// TIA Portal V17 export
// export: Created 2023-12-05T13:40:22.7138877Z, ExportSetting WithDefaults, DisplayName Totally Integrated Automation Portal, DisplayVersion V17, DisplayName TIA Portal Openness, DisplayVersion V17, DisplayName TIA Portal Version Control Interface, DisplayVersion V17, DisplayName SINAMICS Startdrive Advanced, DisplayVersion V17, DisplayName SINAMICS Startdrive G130, G150, S120, S150, SINAMICS MV, S210, DisplayVersion V17, DisplayName SINAMICS Startdrive G110M, G120, G120C, G120D, G120P, G115D, DisplayVersion V17, DisplayName STEP 7 Professional, DisplayVersion V17, DisplayName STEP 7 Safety, DisplayVersion V17, DisplayName WinCC Professional, DisplayVersion V17
FUNCTION "FC531 ACSPN_V5_1_7 Alarms" : Void   // FC531, LAD
{ S7_Optimized_Access := 'TRUE' }
VERSION : 0.1
// LG 16.03.2023 => Changed Slug sensor ON constantly on unit
// LG 30.06.2022 => Changed name of the block (structures are the same like in STD Block V 5_1_6)
// 07.05.2020 => added copying of one alarm from unit IDB (Address DBX74.6) which is new in SB V_5_1_0
// 10.06.2020 => delete 2byte spare (load dbx74.0 to dbx2.0 etc.)
// 08.09.2021 => Changed name of the block (structures are the same like in STD Block V 5_1_0)
// stored: AutoNumber false, IsIECCheckEnabled false, SetENOAutomatically false, UDAEnableTagReadback false
   VAR_INPUT
      "SB DB" : Int;
      "Alarm DB" : Int;
      "Alarm Offset" : Int;
   END_VAR
   VAR_TEMP
      "SB DBW" : Word;
      "AL DBW" : Word;
      "TR DBW" : Word;
   END_VAR
BEGIN

NETWORK
TITLE = Initialization
      L     #"SB DB";
      T     #"SB DBW";
      L     #"Alarm DB";
      T     #"AL DBW";
      L     #"Alarm Offset";
      SLD   3;
      LAR1;

NETWORK
TITLE = Cylinder faults
      CLR;
      OPN   DB [#"SB DBW"];
      L     %DBB70;
      OPN   DB [#"AL DBW"];
      T     DBB [AR1, P#0.0];

NETWORK
TITLE = Cylinder faults
      CLR;
      OPN   DB [#"SB DBW"];
      A     %DBX71.0;
      OPN   DB [#"AL DBW"];
      =     DBX [AR1, P#1.0];

NETWORK
TITLE = RCFaults .0
      CLR;
      OPN   DB [#"SB DBW"];
      A     %DBX74.0;
      OPN   DB [#"AL DBW"];
      =     DBX [AR1, P#4.0];

NETWORK
TITLE = RCFaults .1
      CLR;
      OPN   DB [#"SB DBW"];
      A     %DBX74.1;
      OPN   DB [#"AL DBW"];
      =     DBX [AR1, P#4.1];

NETWORK
TITLE = RCFaults .2
      CLR;
      OPN   DB [#"SB DBW"];
      A     %DBX74.2;
      OPN   DB [#"AL DBW"];
      =     DBX [AR1, P#2.2];

NETWORK
TITLE = RCFaults .3
      CLR;
      OPN   DB [#"SB DBW"];
      A     %DBX74.3;
      OPN   DB [#"AL DBW"];
      =     DBX [AR1, P#4.3];

NETWORK
TITLE = RCFaults .4
      CLR;
      OPN   DB [#"SB DBW"];
      A     %DBX74.4;
      OPN   DB [#"AL DBW"];
      =     DBX [AR1, P#4.4];

NETWORK
TITLE = RCFaults .5
      CLR;
      OPN   DB [#"SB DBW"];
      A     %DBX74.5;
      OPN   DB [#"AL DBW"];
      =     DBX [AR1, P#4.5];

NETWORK
TITLE = RCFaults .6
      CLR;
      OPN   DB [#"SB DBW"];
      A     %DBX74.6;
      OPN   DB [#"AL DBW"];
      =     DBX [AR1, P#4.6];

NETWORK
TITLE = Faults .0
      CLR;
      OPN   DB [#"SB DBW"];
      A     %DBX76.0;
      OPN   DB [#"AL DBW"];
      =     DBX [AR1, P#6.0];

NETWORK
TITLE = Faults .1
      CLR;
      OPN   DB [#"SB DBW"];
      A     %DBX76.1;
      OPN   DB [#"AL DBW"];
      =     DBX [AR1, P#5.6];

NETWORK
TITLE = Faults .2
      CLR;
      OPN   DB [#"SB DBW"];
      A     %DBX76.2;
      OPN   DB [#"AL DBW"];
      =     DBX [AR1, P#6.2];

NETWORK
TITLE = Faults .3
      CLR;
      OPN   DB [#"SB DBW"];
      A     %DBX76.3;
      OPN   DB [#"AL DBW"];
      =     DBX [AR1, P#6.3];

NETWORK
TITLE = Faults .4
      CLR;
      OPN   DB [#"SB DBW"];
      A     %DBX76.4;
      OPN   DB [#"AL DBW"];
      =     DBX [AR1, P#6.4];
END_FUNCTION
